# EPICS autosave request: iocBoot/ioc13MeasCompETC_1/auto_settings.req
file "ETC_settings.req", P=13ETC_1:
